Yaskawa INFORM job: SKRZYNIA_5040_180_STOPNI_20BR.JBI

/JOB
//NAME SKRZYNIA_5040_180_STOPNI_20BR
///FOLDERNAME 02-SKRZYNIE_JOBS
//POS
///NPOS 317,317,0,20,0,0
///TOOL 0
///POSTYPE PULSE
///PULSE
C00000=2424,-36726,63513,-9090,2744,5131
C00001=17840,-61498,-6635,149088,-29435,16513
C00002=84284,-61498,-6635,149088,14842,16513
C00003=84426,-61498,-62039,149088,14842,16513
C00004=84426,-61498,-83719,149088,14842,16513
C00005=79414,-27317,-83719,149088,18958,2543
C00006=73372,-22345,-79926,156833,908,-5737
C00007=69654,-19285,-77591,161600,-10201,-10832
C00008=80044,-19258,-92768,151274,-43492,-95
C00009=80167,-17748,-91560,151286,-43793,-146
C00010=77855,-16084,-90189,153542,-43693,-832
C00011=79745,-14573,-88908,151903,-44240,-404
C00012=80167,-17748,-91560,151286,-43793,-146
C00013=69654,-19285,-77591,161600,-10201,-10832
C00014=57344,-27370,-54568,135214,21884,-6631
C00015=40625,-29987,-49847,90639,36967,7668
C00016=40625,-29987,-49847,90639,36967,7668
C00017=38826,-24689,-45962,89185,38103,8693
C00018=37513,-22163,-43982,88710,38957,9107
C00019=39668,-21791,-43686,88310,37528,9139
C00020=38826,-24689,-45962,89185,38103,8693
C00021=38826,-24689,-45962,89185,38103,8693
C00022=42409,-29700,-46133,101604,34212,3947
C00023=39533,-32421,-42056,71487,38902,9246
C00024=48036,-29192,-45512,38244,44119,19118
C00025=48294,-22040,-40120,37064,45319,19886
C00026=46721,-19694,-38209,37780,46327,19540
C00027=48498,-19279,-37864,36630,45652,20159
C00028=48294,-22040,-40120,37064,45319,19886
C00029=39533,-32421,-42056,71487,38902,9246
C00030=80982,-65498,-53595,111483,16829,-11863
C00031=83918,-61953,-48743,149551,29621,-25735
C00032=40577,-31455,-39147,101508,36831,1521
C00033=62120,-15586,-68046,125419,11390,483
C00034=60388,-9931,-64401,116490,11174,5090
C00035=60671,-7045,-63303,110274,10395,8002
C00036=59274,-5305,-61557,108886,11033,8950
C00037=60834,-4584,-60819,109690,10258,8249
C00038=60671,-7045,-63303,110274,10395,8002
C00039=63645,-11488,-68603,127053,9270,213
C00040=46424,-32589,-51504,107545,30005,2440
C00041=40681,-36168,-63553,67140,38442,15724
C00042=40938,-28250,-58216,64472,39150,17313
C00043=40029,-26609,-57013,64509,39850,17414
C00044=42034,-26290,-56776,63350,38705,17844
C00045=40938,-28250,-58216,64472,39150,17313
C00046=45508,-32760,-62864,41083,46895,21518
C00047=52894,-26615,-39300,28664,42870,21364
C00048=47235,-10440,-23632,29897,60724,24736
C00049=57477,-15037,-17222,22818,38920,22189
C00050=55882,-13164,-15543,23879,39595,21547
C00051=57525,-12586,-15014,22628,39205,22306
C00052=57477,-15037,-17222,22818,38920,22189
C00053=51366,-27458,-41337,29323,44055,21022
C00054=95860,-54197,-56233,-11506,28414,43359
C00055=86028,-64310,-60026,34123,6588,25352
C00056=86028,-64310,-60026,34123,6588,25352
C00057=40577,-31455,-39147,101508,36831,1521
C00058=51132,-28512,-40196,130224,31508,-6645
C00059=50713,-22313,-35527,128251,30719,-5539
C00060=49231,-20302,-33901,126844,31206,-4688
C00061=50925,-19906,-33576,127815,30296,-5311
C00062=50713,-22313,-35527,128251,30719,-5539
C00063=49451,-30533,-41612,129729,32711,-6303
C00064=40577,-31455,-39147,101508,36831,1521
C00065=40577,-27956,-24714,110033,39226,-3600
C00066=40286,-31815,-40383,67790,38842,9831
C00067=40401,-25839,-36160,65987,39341,10928
C00068=39238,-23870,-34666,65921,40243,11019
C00069=41502,-23454,-34345,64975,38856,11500
C00070=40401,-25839,-36160,65987,39341,10928
C00071=40577,-31455,-39147,101508,36831,1521
C00072=86028,-64310,-60026,34123,6588,25352
C00073=86028,-64310,-60026,57978,24772,25352
C00074=86028,-64309,-60028,57978,24769,25352
C00075=40577,-31455,-39147,101508,36831,1521
C00076=38903,-31338,-35872,81629,38108,5349
C00077=39925,-26217,-33347,78892,37684,6977
C00078=38254,-23236,-30426,78887,38846,7020
C00079=40125,-23024,-30182,78580,37583,7157
C00080=39925,-26217,-33347,78892,37684,6977
C00081=73009,-49204,-27678,59140,12738,9351
C00082=45844,-59376,-6382,28358,16063,-8083
C00083=0,-52280,40443,0,6876,0
C00084=0,-39497,64868,0,-320,0
C00085=-26447,-43949,27117,-136096,-23097,-25575
C00086=-84284,-61498,-6635,-149088,14842,-16513
C00087=-84426,-61498,-62039,-149088,14842,-16513
C00088=-84426,-61498,-83719,-149088,14842,-16513
C00089=-80044,-19258,-92768,-151274,-43492,95
C00090=-80749,-16896,-90804,-150801,-44007,28
C00091=-79084,-15727,-89832,-152410,-43912,514
C00092=-80653,-14642,-88911,-151047,-44347,160
C00093=-80749,-16896,-90804,-150801,-44007,28
C00094=-75682,-33870,-78741,-101873,-8535,-10935
C00095=-48995,-37760,-57128,-94978,29787,-5634
C00096=-40649,-29976,-49851,-90623,36950,-7675
C00097=-40649,-29976,-49851,-90623,36950,-7675
C00098=-40401,-23900,-45312,-88796,37053,-8777
C00099=-39435,-22127,-43911,-88459,37683,-9068
C00100=-40828,-22111,-43897,-88252,36759,-9057
C00101=-40401,-23900,-45312,-88796,37053,-8777
C00102=-38849,-24678,-45965,-89170,38087,-8700
C00103=-42432,-29691,-46140,-101591,34194,-3953
C00104=-39561,-32409,-42051,-71473,38885,-9254
C00105=-48061,-29176,-45495,-38229,44108,-19126
C00106=-49260,-20540,-32676,-39004,41808,-18545
C00107=-48004,-18750,-31193,-39572,42610,-18251
C00108=-49371,-18582,-31053,-38688,42033,-18742
C00109=-49260,-20540,-32676,-39004,41808,-18545
C00110=-39561,-30849,-34727,-76036,37950,-6495
C00111=-96080,-64740,-46265,-152525,12897,30451
C00112=-81019,-62154,-45781,-119230,18197,15675
C00113=-39561,-30849,-34727,-76036,37950,-6495
C00114=-48406,-29556,-69320,-92179,25398,-12686
C00115=-47328,-23620,-66389,-87519,25941,-15295
C00116=-49848,-19619,-64817,-82594,24521,-17422
C00117=-48924,-18187,-63619,-82477,25084,-17649
C00118=-50351,-17944,-63415,-81734,24256,-17779
C00119=-49848,-19619,-64817,-82594,24521,-17422
C00120=-49519,-27286,-70984,-91916,23952,-13794
C00121=-40751,-34689,-48106,-81426,35657,-8146
C00122=-40681,-36168,-63553,-67140,38442,-15724
C00123=-43821,-29034,-57028,-64528,36876,-16908
C00124=-42088,-26142,-54916,-64622,38193,-17071
C00125=-43742,-25965,-54783,-63683,37230,-17421
C00126=-43821,-29034,-57028,-64528,36876,-16908
C00127=-45534,-32689,-56736,-43795,43869,-19675
C00128=-52916,-25303,-32096,-30881,39442,-19966
C00129=-58280,-19120,-27405,-20546,42356,-23593
C00130=-59518,-12125,-8161,-23315,34652,-21915
C00131=-57886,-10293,-6452,-24525,35301,-21178
C00132=-59048,-10070,-6241,-23572,34987,-21754
C00133=-59518,-12125,-8161,-23315,34652,-21915
C00134=-51388,-26224,-34221,-31487,40653,-19631
C00135=-51388,-26224,-34221,-31487,40653,-19631
C00136=-88798,-58761,-51280,2265,16070,-39336
C00137=-86028,-64310,-60026,-34123,6588,-25352
C00138=-40577,-31455,-39147,-101508,36831,-1521
C00139=-51132,-28512,-40196,-130224,31508,6645
C00140=-53828,-21538,-34856,-130236,29103,6776
C00141=-52017,-19235,-32968,-128427,29694,5703
C00142=-53263,-19086,-32845,-129254,29059,6216
C00143=-53828,-21538,-34856,-130236,29103,6776
C00144=-49451,-30533,-41612,-129729,32711,6303
C00145=-40577,-31455,-39147,-101508,36831,-1521
C00146=-40577,-27956,-24714,-110033,39226,3600
C00147=-40286,-31815,-40383,-67790,38842,-9831
C00148=-43936,-25540,-35936,-64541,37153,-11660
C00149=-42305,-23005,-33995,-64547,38400,-11722
C00150=-43835,-22890,-33904,-63890,37459,-12051
C00151=-43936,-25540,-35936,-64541,37153,-11660
C00152=-40577,-31455,-39147,-101508,36831,-1521
C00153=-86028,-64310,-60026,-34123,6588,-25352
C00154=-86028,-64310,-60026,-57978,24772,-25352
C00155=-86028,-64309,-60028,-57978,24769,-25352
C00156=-38903,-32774,-42709,-77257,38620,-7991
C00157=-42184,-24671,-30182,-79828,36015,-6379
C00158=-40569,-22194,-28667,-79025,37222,-6883
C00159=-42422,-21657,-27035,-79658,35870,-6476
C00160=-42184,-24671,-30182,-79828,36015,-6379
C00161=-49485,-27068,-14424,-72878,29346,-3454
C00162=-73009,-40277,-6382,-95546,11240,8083
C00163=-45844,-59376,-6382,-28358,16063,8083
C00164=0,-52280,40443,0,6876,0
C00165=-328,-40297,61840,-3808,1166,2006
C00166=17840,-61498,-6635,149088,-29435,16513
C00167=84284,-61498,-6635,149088,14842,16513
C00168=84513,-69641,-44219,158038,21366,7151
C00169=47085,-54494,-58070,115522,48054,-5105
C00170=38967,-30574,-72694,69596,39131,19833
C00171=38967,-30574,-72694,69596,39131,19833
C00172=40878,-31428,-43525,94415,35447,4548
C00173=41854,-23003,-37366,91536,34575,6162
C00174=41898,-23706,-43940,85918,34440,9382
C00175=40878,-31428,-43525,94415,35447,4548
C00176=39533,-30860,-34732,76047,37967,6488
C00177=46634,-28948,-39362,44629,40673,16329
C00178=47197,-19209,-31862,42612,41940,17576
C00179=47198,-18019,-24610,45914,39068,15513
C00180=46634,-28948,-39362,44629,40673,16329
C00181=49331,-35046,-41363,50989,36464,13786
C00182=89354,-53419,-27647,126582,13574,2293
C00183=87455,-53096,-27566,122620,14401,3981
C00184=17840,-61498,-6635,149088,-29435,16513
C00185=0,-40660,62594,0,368,0
C00186=-17840,-45374,24451,-139252,-21484,-21626
C00187=-84284,-61498,-6635,-149088,14842,-16513
C00188=-72689,-59179,-38530,-131034,19974,-20147
C00189=-60772,-50498,-67929,-131953,39604,8737
C00190=-35436,-23032,-76859,-79659,38842,-23552
C00191=-45272,-23185,-79217,-69622,29986,-24621
C00192=-40692,-30585,-47134,-93878,35604,-6100
C00193=-40001,-32873,-51156,-81642,36602,-9590
C00194=-40001,-32873,-51156,-81642,36602,-9590
C00195=-40670,-20516,-31954,-95909,37519,2638
C00196=-40659,-21415,-38860,-90776,37084,-418
C00197=-40001,-32873,-51156,-81642,36602,-9590
C00198=-40870,-31947,-42232,-63836,39356,-11267
C00199=-49698,-28191,-44773,-34393,44991,-20180
C00200=-50470,-17992,-36746,-32748,46471,-21232
C00201=-50479,-17271,-29967,-35030,43083,-19704
C00202=-49698,-28191,-44773,-34393,44991,-20180
C00203=-49698,-28786,-61181,-29564,54118,-23727
C00204=-82387,-65169,-54524,-93566,14000,4306
C00205=-84284,-61498,-6635,-149088,14842,-16513
C00206=-17840,-55538,4678,-146289,-26509,-18006
C00207=0,-39879,64121,0,-95,0
C00208=0,-52280,40443,0,6876,0
C00209=0,-52279,40442,0,6873,-1
C00210=65212,-60046,-8049,104848,-4690,-17864
C00211=39533,-30860,-34732,76047,37967,6488
C00212=40614,-18402,-49700,108061,37841,3104
C00213=40614,-18402,-49700,108061,37841,3104
C00214=41485,-12828,-44769,107158,37037,3517
C00215=41606,-12003,-50092,101801,35658,6646
C00216=40614,-18402,-49700,108061,37841,3104
C00217=40614,-18402,-49700,108061,37841,3104
C00218=49502,-29076,-56400,114238,27233,2182
C00219=40723,-34700,-48106,81442,35674,8138
C00220=40409,-20441,-6217,113220,40048,-7375
C00221=42493,-16023,-2566,113375,38437,-7307
C00222=42407,-18778,-11657,108563,36754,-4436
C00223=40409,-20441,-6217,113220,40048,-7375
C00224=39142,-35162,-55050,69516,38837,12809
C00225=56371,-25167,-46588,19640,50472,24717
C00226=56370,-24708,-41585,20550,47569,24051
C00227=56918,-11874,-10453,25192,36609,21079
C00228=55886,-6496,-6457,23354,43942,22802
C00229=56370,-20008,-17514,26362,35642,20382
C00230=64715,-29320,-15625,38703,25818,15298
C00231=92185,-54275,-12566,86648,-10406,-3964
C00232=0,-52279,40442,0,6873,-1
C00233=0,-52279,40442,0,6873,1
C00234=-37964,-53933,3758,-67381,6079,8710
C00235=-49904,-54659,-13207,-92831,9076,10998
C00236=-40577,-31455,-39147,-101508,36831,-1521
C00237=-37616,-19376,-56763,-96336,39614,-8284
C00238=-37616,-19376,-56763,-96336,39614,-8284
C00239=-40511,-13581,-51709,-94759,37718,-8730
C00240=-40499,-12353,-56710,-89299,37353,-11996
C00241=-37616,-19376,-56763,-96336,39614,-8284
C00242=-29868,-22288,-62791,-69139,55102,-14753
C00243=-38799,-34785,-68031,-65062,42004,-17700
C00244=-40843,-35617,-55345,-69003,37714,-12979
C00245=-40440,-20436,-6228,-113223,40025,7374
C00246=-44187,-15892,-2555,-114126,37382,7633
C00247=-44098,-18576,-11485,-109220,35681,4746
C00248=-40440,-20436,-6228,-113223,40025,7374
C00249=-39177,-35147,-55048,-69491,38818,-12821
C00250=-56396,-25146,-46559,-19625,50462,-24726
C00251=-56395,-19986,-17482,-26346,35629,-20392
C00252=-58275,-11034,-9655,-24079,36290,-21752
C00253=-53190,-4481,-3595,-29275,45221,-22163
C00254=-57665,-14024,-8618,-26361,33798,-20418
C00255=-54116,-36015,-20945,-72642,23963,-3174
C00256=-66633,-56546,-10672,-107930,-1326,17731
C00257=0,-52279,40442,0,6873,1
C00258=1,-52278,40440,0,6869,2
C00259=71244,-62242,-42760,28259,6636,20995
C00260=86028,-64310,-60026,34123,6588,25352
C00261=40577,-31455,-39147,101508,36831,1521
C00262=59968,-20268,-35682,154489,33643,-14406
C00263=49575,-29432,-40732,125662,31704,-5163
C00264=49462,-20616,-33510,124217,30834,-4171
C00265=49522,-21549,-40421,118611,28458,-1132
C00266=49575,-29432,-40732,125662,31704,-5163
C00267=40577,-31455,-39147,101508,36831,1521
C00268=40577,-27956,-24714,110033,39226,-3600
C00269=40745,-32658,-46054,62068,40241,12517
C00270=41807,-24195,-39992,59384,40616,14125
C00271=41807,-23141,-33009,63548,38813,11557
C00272=40745,-32658,-46054,62068,40241,12517
C00273=40577,-31455,-39147,101508,36831,1521
C00274=86028,-64310,-60026,34123,6588,25352
C00275=71244,-62242,-42760,28259,6636,20995
C00276=1,-52278,40440,0,6869,2
C00277=-71244,-62242,-42760,-28259,6636,-20995
C00278=-86028,-64310,-60026,-34123,6588,-25352
C00279=-40577,-31455,-39147,-101508,36831,-1521
C00280=-59968,-20268,-35682,-154489,33643,14406
C00281=-49575,-29432,-40732,-125662,31704,5163
C00282=-51745,-20083,-33073,-125482,29566,4973
C00283=-51720,-20470,-39541,-119439,27111,1736
C00284=-49575,-29432,-40732,-125662,31704,5163
C00285=-40577,-31455,-39147,-101508,36831,-1521
C00286=-40577,-27956,-24714,-110033,39226,3600
C00287=-40745,-32658,-46054,-62068,40241,-12517
C00288=-43918,-23250,-39259,-58141,39481,-14752
C00289=-43886,-22328,-32371,-62491,37605,-12114
C00290=-40745,-32658,-46054,-62068,40241,-12517
C00291=-40577,-31455,-39147,-101508,36831,-1521
C00292=-86028,-64310,-60026,-34123,6588,-25352
C00293=-71244,-62242,-42760,-28259,6636,-20995
C00294=-1,-52278,40440,0,6869,-2
C00295=2,-52272,40438,1,6859,6
C00296=86028,-64309,-60028,57978,24769,25352
C00297=40577,-29271,-29688,107326,38311,-1954
C00298=39686,-18672,-6528,106229,39889,-5106
C00299=40115,-16641,-6285,104879,39175,-4249
C00300=40039,-18622,-13956,100467,38186,-1572
C00301=40578,-24372,-18301,102198,38163,-2598
C00302=51067,-26075,-7125,86189,26964,-2285
C00303=73009,-40277,-6382,95546,11240,-8083
C00304=45844,-59376,-6382,28358,16063,-8083
C00305=0,-52280,40443,0,6876,0
C00306=-49336,-60774,-21138,-33872,18352,-14728
C00307=-86028,-64309,-60028,-57978,24769,-25352
C00308=-40577,-31455,-39147,-101508,36831,-1521
C00309=-39686,-19839,-10359,-104288,39330,3911
C00310=-42399,-15880,-6496,-104843,37485,4096
C00311=-42423,-18479,-15943,-99204,36274,759
C00312=-40581,-27576,-30519,-94819,36955,-1807
C00313=-56174,-25706,-11107,-56673,25485,-9093
C00314=-73009,-40277,-6382,-95546,11240,8083
C00315=-45844,-59376,-6382,-28358,16063,8083
C00316=0,-52280,40443,0,6876,0
BC00000=467540
BC00001=467540
BC00002=467540
BC00003=467540
BC00004=467540
BC00005=467540
BC00006=467540
BC00007=467540
BC00008=467540
BC00009=467540
BC00010=467540
BC00011=467540
BC00012=467540
BC00013=467540
BC00014=507878
BC00015=487125
BC00016=487125
BC00017=487125
BC00018=487125
BC00019=487125
BC00020=487125
BC00021=487125
BC00022=485653
BC00023=485653
BC00024=485653
BC00025=485653
BC00026=485653
BC00027=485653
BC00028=485653
BC00029=485653
BC00030=485653
BC00031=675626
BC00032=675626
BC00033=714617
BC00034=714617
BC00035=714617
BC00036=714617
BC00037=714617
BC00038=714617
BC00039=717870
BC00040=686402
BC00041=686402
BC00042=686402
BC00043=686402
BC00044=686402
BC00045=686402
BC00046=655680
BC00047=655680
BC00048=655680
BC00049=655680
BC00050=655680
BC00051=655680
BC00052=655680
BC00053=612974
BC00054=633023
BC00055=817027
BC00056=849627
BC00057=849627
BC00058=849627
BC00059=849627
BC00060=849627
BC00061=849627
BC00062=849627
BC00063=849627
BC00064=849627
BC00065=849627
BC00066=849627
BC00067=849627
BC00068=849627
BC00069=849627
BC00070=849627
BC00071=849627
BC00072=849627
BC00073=849627
BC00074=994223
BC00075=997528
BC00076=995174
BC00077=996484
BC00078=995671
BC00079=995573
BC00080=996484
BC00081=965704
BC00082=879640
BC00083=828403
BC00084=484492
BC00085=467540
BC00086=467540
BC00087=467540
BC00088=467540
BC00089=467540
BC00090=467542
BC00091=467542
BC00092=467542
BC00093=467542
BC00094=476933
BC00095=486269
BC00096=487125
BC00097=487125
BC00098=487125
BC00099=487125
BC00100=487125
BC00101=487125
BC00102=487125
BC00103=485653
BC00104=485653
BC00105=485653
BC00106=477973
BC00107=477973
BC00108=477973
BC00109=477973
BC00110=477973
BC00111=477973
BC00112=637224
BC00113=637224
BC00114=676215
BC00115=676215
BC00116=676215
BC00117=676215
BC00118=676215
BC00119=676215
BC00120=679468
BC00121=648000
BC00122=686402
BC00123=686402
BC00124=686402
BC00125=686402
BC00126=686402
BC00127=648000
BC00128=648000
BC00129=648000
BC00130=648000
BC00131=648000
BC00132=648000
BC00133=648000
BC00134=648000
BC00135=624365
BC00136=626985
BC00137=849627
BC00138=849627
BC00139=849627
BC00140=849627
BC00141=849627
BC00142=849627
BC00143=849627
BC00144=849627
BC00145=849627
BC00146=849627
BC00147=849627
BC00148=849627
BC00149=849627
BC00150=849627
BC00151=849627
BC00152=849627
BC00153=849627
BC00154=849627
BC00155=994094
BC00156=1002378
BC00157=995010
BC00158=995501
BC00159=994027
BC00160=995010
BC00161=965704
BC00162=944514
BC00163=879640
BC00164=828403
BC00165=489545
BC00166=498510
BC00167=467540
BC00168=484470
BC00169=489677
BC00170=489675
BC00171=489675
BC00172=477973
BC00173=477973
BC00174=477973
BC00175=477973
BC00176=477973
BC00177=477973
BC00178=477973
BC00179=477973
BC00180=477973
BC00181=458600
BC00182=448949
BC00183=525722
BC00184=487426
BC00185=486611
BC00186=479113
BC00187=467540
BC00188=470459
BC00189=528079
BC00190=528079
BC00191=528077
BC00192=477973
BC00193=477973
BC00194=477973
BC00195=477973
BC00196=477973
BC00197=477973
BC00198=477973
BC00199=477973
BC00200=477973
BC00201=477973
BC00202=477973
BC00203=477973
BC00204=477973
BC00205=467540
BC00206=467540
BC00207=482699
BC00208=527850
BC00209=541981
BC00210=560285
BC00211=642547
BC00212=672480
BC00213=672480
BC00214=672480
BC00215=672480
BC00216=672480
BC00217=672480
BC00218=679468
BC00219=648000
BC00220=648000
BC00221=648000
BC00222=648000
BC00223=648000
BC00224=648000
BC00225=648000
BC00226=648000
BC00227=648000
BC00228=648000
BC00229=607087
BC00230=565122
BC00231=563264
BC00232=528036
BC00233=500175
BC00234=526377
BC00235=553881
BC00236=649161
BC00237=672480
BC00238=672480
BC00239=672480
BC00240=672480
BC00241=672480
BC00242=634078
BC00243=641066
BC00244=648000
BC00245=648000
BC00246=648000
BC00247=648000
BC00248=648000
BC00249=648000
BC00250=648000
BC00251=608255
BC00252=648000
BC00253=648000
BC00254=613281
BC00255=601855
BC00256=554421
BC00257=532052
BC00258=574254
BC00259=802302
BC00260=849627
BC00261=849627
BC00262=849627
BC00263=849627
BC00264=849627
BC00265=849627
BC00266=849627
BC00267=849627
BC00268=849627
BC00269=849627
BC00270=849627
BC00271=849627
BC00272=849627
BC00273=849627
BC00274=849627
BC00275=802302
BC00276=652677
BC00277=802302
BC00278=849627
BC00279=849627
BC00280=849627
BC00281=849627
BC00282=849627
BC00283=849627
BC00284=849627
BC00285=849627
BC00286=849627
BC00287=849627
BC00288=849627
BC00289=849627
BC00290=849627
BC00291=849627
BC00292=849627
BC00293=802302
BC00294=652677
BC00295=780547
BC00296=1007134
BC00297=993409
BC00298=989933
BC00299=991571
BC00300=991571
BC00301=990663
BC00302=974575
BC00303=965704
BC00304=879640
BC00305=828403
BC00306=894245
BC00307=994909
BC00308=994105
BC00309=993208
BC00310=992554
BC00311=992554
BC00312=984659
BC00313=957065
BC00314=965704
BC00315=879640
BC00316=828403
///POSTYPE BASE
///RECTAN
///RCONF 1,0,0,0,0,0,0,0,0,0,0,0,0,0,0,0,0,0,0,0,0,0,0,0
P00006=0.000,0.000,0.000,0.0000,0.0000,0.0000
///RCONF 0,0,0,0,0,0,0,0,0,0,0,0,0,0,0,0,0,0,0,0,0,0,0,0
P00056=0.000,0.000,5.000,0.0000,0.0000,0.0000
///RCONF 1,0,0,0,0,0,0,0,0,0,0,0,0,0,0,0,0,0,0,0,0,0,0,0
P00300=-0.036,-1.505,2.318,0.0000,0.0000,0.0000
P00301=0.028,-0.041,7.752,0.0000,0.0000,0.0000
///RCONF 0,0,0,0,0,0,0,0,0,0,0,0,0,0,0,0,0,0,0,0,0,0,0,0
P00302=0.052,-2.937,-4.426,0.0000,0.0000,0.0000
P00303=-0.004,-1.437,-4.584,0.0000,0.0000,0.0000
P00304=0.028,-1.666,-4.234,0.0000,0.0000,0.0000
P00305=-0.003,-1.920,-3.501,0.0000,0.0000,0.0000
P00306=0.015,-2.252,-3.054,0.0000,0.0000,0.0000
P00307=0.019,-2.151,-5.077,0.0000,0.0000,0.0000
P00308=-0.003,-2.092,-4.888,0.0000,0.0000,0.0000
P00350=11.519,-0.008,1.149,0.0000,0.0000,0.0000
P00351=13.563,-0.027,-0.653,0.0000,0.0000,0.0000
P00352=13.252,-0.027,-0.827,0.0000,0.0000,0.0000
P00353=10.971,-0.082,0.776,0.0000,0.0000,0.0000
P00354=-0.024,2.508,-1.824,0.0000,0.0000,0.0000
P00355=-0.001,2.528,-1.131,0.0000,0.0000,0.0000
P00356=-0.034,2.921,-0.262,0.0000,0.0000,0.0000
P00357=0.003,3.386,-0.091,0.0000,0.0000,0.0000
P00358=0.014,3.037,-0.020,0.0000,0.0000,0.0000
//INST
///DATE 2024/05/16 17:47
///ATTR SC,RW
///GROUP1 RB1,BS1
NOP
CALL JOB:MOVE_INTO_TUNNEL
MOVJ C00000 BC00000 VJ=10.00
MOVJ C00001 BC00001 VJ=10.00
MOVJ C00002 BC00002 VJ=10.00
MOVJ C00003 BC00003 VJ=10.00
MOVJ C00004 BC00004 VJ=10.00
MOVJ C00005 BC00005 VJ=10.00
MOVJ C00006 BC00006 VJ=10.00
MOVL C00007 BC00007 V=150.0
MOVL C00008 BC00008 V=150.0
'------------------------
'W63.3
'------------------------
MOVL C00009 BC00009 V=66.7 PL=0
REFP 3 C00010 BC00010
CALL JOB:SEARCH-R1
IMOV P0056 V=23.0
SET P0300 P0006
SFTON P0300
REFP 3 C00011 BC00011
CALL JOB:SEARCH-R1
SET P0300 P0006
SFTON P0300
MOVL C00012 BC00012 V=66.7 PL=0
SFTOF
'PRZEJAZD
MOVL C00013 BC00013 V=150.0
MOVL C00014 BC00014 V=666.7
MOVJ C00015 BC00015 VJ=10.00
MOVL C00016 BC00016 V=150.0
'------------------------
'W29.6
'------------------------
MOVL C00017 BC00017 V=66.7 PL=0
REFP 3 C00018 BC00018
CALL JOB:SEARCH-R1
IMOV P0056 V=23.0 PL=0
SET P0301 P0006
SFTON P0301
REFP 3 C00019 BC00019
CALL JOB:SEARCH-R1
SET P0301 P0006
SFTON P0301
MOVL C00020 BC00020 V=66.7 PL=0
SFTOF
'PRZEJAZD
MOVL C00021 BC00021 V=500.0
MOVL C00022 BC00022 V=500.0
MOVL C00023 BC00023 V=500.0
MOVL C00024 BC00024 V=500.0
'------------------------
'W29.9
'------------------------
MOVL C00025 BC00025 V=66.7 PL=0
REFP 3 C00026 BC00026
CALL JOB:SEARCH-R1
IMOV P0056 V=23.0 PL=0
SET P0302 P0006
SFTON P0302
REFP 3 C00027 BC00027
CALL JOB:SEARCH-R1
SET P0302 P0006
SFTON P0302
MOVL C00028 BC00028 V=66.7 PL=0
SFTOF
MOVL C00029 BC00029 V=500.0
'PRZEJAZD
MOVL C00030 BC00030 V=500.0
MOVJ C00031 BC00031 VJ=10.00
MOVL C00032 BC00032 V=500.0
MOVL C00033 BC00033 V=500.0
MOVL C00034 BC00034 V=500.0
'------------------------
'W63.12
'------------------------
MOVL C00035 BC00035 V=66.7 PL=0
REFP 3 C00036 BC00036
CALL JOB:SEARCH-R1
IMOV P0056 V=23.0 PL=0
SET P0303 P0006
SFTON P0303
REFP 3 C00037 BC00037
CALL JOB:SEARCH-R1
SET P0303 P0006
SFTON P0303
MOVL C00038 BC00038 V=66.7 PL=0
SFTOF
'PRZEJAZD
MOVL C00039 BC00039 V=500.0
MOVL C00040 BC00040 V=500.0
MOVL C00041 BC00041 V=500.0
'------------------------
'W63.15
'------------------------
MOVL C00042 BC00042 V=66.7 PL=0
REFP 3 C00043 BC00043
CALL JOB:SEARCH-R1
IMOV P0056 V=23.0 PL=0
SET P0304 P0006
SFTON P0304
REFP 3 C00044 BC00044
CALL JOB:SEARCH-R1
SET P0304 P0006
SFTON P0304
MOVL C00045 BC00045 V=66.7 PL=0
SFTOF
'PRZEJAZD
MOVL C00046 BC00046 V=500.0
MOVL C00047 BC00047 V=500.0
MOVL C00048 BC00048 V=500.0
'------------------------
'W29.18
'------------------------
MOVL C00049 BC00049 V=66.7 PL=0
REFP 3 C00050 BC00050
CALL JOB:SEARCH-R1
IMOV P0056 V=23.0 PL=0
SET P0305 P0006
SFTON P0305
REFP 3 C00051 BC00051
CALL JOB:SEARCH-R1
SET P0305 P0006
SFTON P0305
MOVL C00052 BC00052 V=66.7 PL=0
SFTOF
'PRZEJAZD
MOVL C00053 BC00053 V=500.0
MOVJ C00054 BC00054 VJ=10.00
MOVJ C00055 BC00055 VJ=10.00
MOVJ C00056 BC00056 VJ=10.00
MOVL C00057 BC00057 V=500.0
MOVL C00058 BC00058 V=500.0
'------------------------
'W29.21
'------------------------
MOVL C00059 BC00059 V=66.7 PL=0
REFP 3 C00060 BC00060
CALL JOB:SEARCH-R1
IMOV P0056 V=23.0 PL=0
SET P0306 P0006
SFTON P0306
REFP 3 C00061 BC00061
CALL JOB:SEARCH-R1
SET P0306 P0006
SFTON P0306
MOVL C00062 BC00062 V=66.7 PL=0
SFTOF
'PRZEJAZD
MOVL C00063 BC00063 V=500.0
MOVL C00064 BC00064 V=500.0
MOVL C00065 BC00065 V=500.0
MOVL C00066 BC00066 V=500.0
'------------------------
'W29.24
'------------------------
MOVL C00067 BC00067 V=66.7 PL=0
REFP 3 C00068 BC00068
CALL JOB:SEARCH-R1
IMOV P0056 V=23.0 PL=0
SET P0307 P0006
SFTON P0307
REFP 3 C00069 BC00069
CALL JOB:SEARCH-R1
SET P0307 P0006
SFTON P0307
MOVL C00070 BC00070 V=66.7 PL=0
SFTOF
'PRZEJAZD
MOVL C00071 BC00071 V=500.0
MOVL C00072 BC00072 V=500.0
MOVL C00073 BC00073 V=500.0
MOVL C00074 BC00074 V=500.0
MOVL C00075 BC00075 V=500.0
MOVL C00076 BC00076 V=500.0
'BRAK MOZLIWOSCI 29.27
'BRAK MOZLIWOSCI 29.27
'BRAK MOZLIWOSCI 29.27
'BRAK MOZLIWOSCI 29.27
'BRAK MOZLIWOSCI 29.27
'------------------------
'W63.30
'------------------------
MOVL C00077 BC00077 V=166.7 PL=0
REFP 3 C00078 BC00078
CALL JOB:SEARCH-R1
IMOV P0056 V=23.0 PL=0
SET P0308 P0006
SFTON P0308
REFP 3 C00079 BC00079
CALL JOB:SEARCH-R1
SET P0308 P0006
SFTON P0308
MOVL C00080 BC00080 V=250.0 PL=0
SFTOF
'PRZEJAZD
MOVJ C00081 BC00081 VJ=20.00
MOVJ C00082 BC00082 VJ=30.00
MOVJ C00083 BC00083 VJ=30.00
MOVJ C00084 BC00084 VJ=40.00
MOVJ C00085 BC00085 VJ=20.00
MOVJ C00086 BC00086 VJ=20.00
MOVJ C00087 BC00087 VJ=20.00
MOVJ C00088 BC00088 VJ=20.00
MOVL C00089 BC00089 V=500.0
'------------------------
'W63.3
'------------------------
MOVL C00090 BC00090 V=66.7 PL=0
REFP 3 C00091 BC00091
CALL JOB:SEARCH-R1
IMOV P0056 V=23.0
SET P0350 P0006
SFTON P0350
REFP 3 C00092 BC00092
CALL JOB:SEARCH-R1
SET P0350 P0006
SFTON P0350
MOVL C00093 BC00093 V=66.7 PL=0
SFTOF
'PRZEJAZD
MOVL C00094 BC00094 V=150.0 PL=0
MOVJ C00095 BC00095 VJ=10.00
MOVJ C00096 BC00096 VJ=10.00
MOVL C00097 BC00097 V=150.0
'------------------------
'W29.6
'------------------------
MOVL C00098 BC00098 V=66.7 PL=0
REFP 3 C00099 BC00099
CALL JOB:SEARCH-R1
IMOV P0056 V=23.0 PL=0
SET P0351 P0006
SFTON P0351
REFP 3 C00100 BC00100
CALL JOB:SEARCH-R1
SET P0351 P0006
SFTON P0351
MOVL C00101 BC00101 V=66.7 PL=0
SFTOF
'PRZEJAZD
MOVL C00102 BC00102 V=500.0
MOVL C00103 BC00103 V=500.0
MOVL C00104 BC00104 V=500.0
MOVL C00105 BC00105 V=500.0
'------------------------
'W29.9
'------------------------
MOVL C00106 BC00106 V=66.7 PL=0
REFP 3 C00107 BC00107
CALL JOB:SEARCH-R1
IMOV P0056 V=23.0 PL=0
SET P0352 P0006
SFTON P0352
REFP 3 C00108 BC00108
CALL JOB:SEARCH-R1
SET P0352 P0006
SFTON P0352
MOVL C00109 BC00109 V=66.7 PL=0
SFTOF
MOVL C00110 BC00110 V=500.0
'PRZEJAZD
MOVL C00111 BC00111 V=500.0
MOVJ C00112 BC00112 VJ=30.00
MOVL C00113 BC00113 V=500.0
MOVL C00114 BC00114 V=500.0
MOVL C00115 BC00115 V=500.0
'------------------------
'W63.12
'------------------------
MOVL C00116 BC00116 V=66.7 PL=0
REFP 3 C00117 BC00117
CALL JOB:SEARCH-R1
IMOV P0056 V=23.0 PL=0
SET P0353 P0006
SFTON P0353
REFP 3 C00118 BC00118
CALL JOB:SEARCH-R1
SET P0353 P0006
SFTON P0353
MOVL C00119 BC00119 V=66.7 PL=0
SFTOF
'PRZEJAZD
MOVL C00120 BC00120 V=500.0
MOVL C00121 BC00121 V=500.0
MOVL C00122 BC00122 V=500.0
'------------------------
'W63.15
'------------------------
MOVL C00123 BC00123 V=66.7 PL=0
REFP 3 C00124 BC00124
CALL JOB:SEARCH-R1
IMOV P0056 V=23.0 PL=0
SET P0354 P0006
SFTON P0354
REFP 3 C00125 BC00125
CALL JOB:SEARCH-R1
SET P0354 P0006
SFTON P0354
MOVL C00126 BC00126 V=66.7 PL=0
SFTOF
'PRZEJAZD
MOVL C00127 BC00127 V=500.0
MOVL C00128 BC00128 V=500.0
MOVL C00129 BC00129 V=500.0
'------------------------
'W29.18
'------------------------
MOVL C00130 BC00130 V=66.7 PL=0
REFP 3 C00131 BC00131
CALL JOB:SEARCH-R1
IMOV P0056 V=23.0 PL=0
SET P0355 P0006
SFTON P0355
REFP 3 C00132 BC00132
CALL JOB:SEARCH-R1
SET P0355 P0006
SFTON P0355
MOVL C00133 BC00133 V=66.7 PL=0
SFTOF
'PRZEJAZD
MOVL C00134 BC00134 V=500.0
MOVJ C00135 BC00135 VJ=10.00
MOVJ C00136 BC00136 VJ=10.00
MOVJ C00137 BC00137 VJ=30.00
MOVL C00138 BC00138 V=500.0
MOVL C00139 BC00139 V=500.0
'------------------------
'W29.21
'------------------------
MOVL C00140 BC00140 V=66.7 PL=0
REFP 3 C00141 BC00141
CALL JOB:SEARCH-R1
IMOV P0056 V=23.0 PL=0
SET P0356 P0006
SFTON P0356
REFP 3 C00142 BC00142
CALL JOB:SEARCH-R1
SET P0356 P0006
SFTON P0356
MOVL C00143 BC00143 V=66.7 PL=0
SFTOF
'PRZEJAZD
MOVL C00144 BC00144 V=500.0
MOVL C00145 BC00145 V=500.0
MOVL C00146 BC00146 V=500.0
MOVL C00147 BC00147 V=500.0
'------------------------
'W29.24
'------------------------
MOVL C00148 BC00148 V=66.7 PL=0
REFP 3 C00149 BC00149
CALL JOB:SEARCH-R1
IMOV P0056 V=23.0 PL=0
SET P0357 P0006
SFTON P0357
REFP 3 C00150 BC00150
CALL JOB:SEARCH-R1
SET P0357 P0006
SFTON P0357
MOVL C00151 BC00151 V=66.7 PL=0
SFTOF
'PRZEJAZD
MOVL C00152 BC00152 V=500.0
MOVL C00153 BC00153 V=500.0
MOVL C00154 BC00154 V=500.0
MOVL C00155 BC00155 V=500.0
MOVL C00156 BC00156 V=500.0
'BRAK MOZLIWOSCI 29.27
'BRAK MOZLIWOSCI 29.27
'BRAK MOZLIWOSCI 29.27
'BRAK MOZLIWOSCI 29.27
'BRAK MOZLIWOSCI 29.27
'------------------------
'W63.30
'------------------------
MOVL C00157 BC00157 V=66.7 PL=0
REFP 3 C00158 BC00158
CALL JOB:SEARCH-R1
IMOV P0056 V=23.0 PL=0
SET P0358 P0006
SFTON P0358
REFP 3 C00159 BC00159
CALL JOB:SEARCH-R1
SET P0358 P0006
SFTON P0358
MOVL C00160 BC00160 V=66.7 PL=0
SFTOF
'PRZEJAZD
MOVL C00161 BC00161 V=500.0
MOVJ C00162 BC00162 VJ=30.00
MOVJ C00163 BC00163 VJ=30.00
MOVJ C00164 BC00164 VJ=30.00
MOVJ C00165 BC00165 VJ=30.00
MOVJ C00166 BC00166 VJ=20.00
MOVJ C00167 BC00167 VJ=20.00
MOVJ C00168 BC00168 VJ=20.00
MOVJ C00169 BC00169 VJ=20.00
SFTOF
'------------------------
'W63.3
'------------------------
'PRZEJAZD
MOVL C00170 BC00170 V=500.0
MOVL C00171 BC00171 V=500.0
'------------------------
'W29.6
'------------------------
MOVL C00172 BC00172 V=500.0
SFTON P0301
MOVL C00173 BC00173 V=166.7 PL=0
MACRO1 MJ#(0) ARGF24
ARCON
MOVL C00174 BC00174 V=10.8
ARCOF
SFTOF
MOVL C00175 BC00175 V=500.0
SFTOF
MOVL C00176 BC00176 V=500.0
'------------------------
'W29.9
'------------------------
MOVL C00177 BC00177 V=500.0
SFTON P0302
MOVL C00178 BC00178 V=66.7 PL=0
MACRO1 MJ#(0) ARGF24
ARCON
MOVL C00179 BC00179 V=10.8
ARCOF
SFTOF
MOVL C00180 BC00180 V=500.0
SFTOF
'PRZEJAZD
MOVL C00181 BC00181 V=500.0
MOVJ C00182 BC00182 VJ=10.00
MOVJ C00183 BC00183 VJ=10.00
MOVJ C00184 BC00184 VJ=10.00
MOVJ C00185 BC00185 VJ=10.00
'TEST
'TEST
'TEST
MOVJ C00186 BC00186 VJ=30.00
MOVJ C00187 BC00187 VJ=10.00
MOVJ C00188 BC00188 VJ=10.00
MOVJ C00189 BC00189 VJ=20.00
MOVL C00190 BC00190 V=500.0
MOVL C00191 BC00191 V=500.0
MOVL C00192 BC00192 V=500.0
MOVL C00193 BC00193 V=500.0
'------------------------
'W28.6
'------------------------
MOVL C00194 BC00194 V=500.0
SFTON P0351
MOVL C00195 BC00195 V=166.7 PL=0
MACRO1 MJ#(0) ARGF24
ARCON
MOVL C00196 BC00196 V=10.8
ARCOF
SFTOF
MOVL C00197 BC00197 V=500.0
SFTOF
MOVL C00198 BC00198 V=500.0
'------------------------
'W28.9
'------------------------
MOVL C00199 BC00199 V=500.0
SFTON P0352
MOVL C00200 BC00200 V=66.7 PL=0
MACRO1 MJ#(0) ARGF24
ARCON
MOVL C00201 BC00201 V=10.0
ARCOF
SFTOF
MOVL C00202 BC00202 V=500.0
SFTOF
'PRZEJAZD
MOVL C00203 BC00203 V=666.7
MOVL C00204 BC00204 V=500.0
MOVJ C00205 BC00205 VJ=10.00
MOVJ C00206 BC00206 VJ=10.00
MOVJ C00207 BC00207 VJ=20.00
MOVJ C00208 BC00208 VJ=30.00
MOVJ C00209 BC00209 VJ=30.00
MOVJ C00210 BC00210 VJ=20.00
MOVJ C00211 BC00211 VJ=20.00
'------------------------
'W63.12
'------------------------
MOVL C00212 BC00212 V=500.0
MOVL C00213 BC00213 V=66.7
SFTON P0303
MOVL C00214 BC00214 V=166.7 PL=0
ARCON
MOVL C00215 BC00215 V=10.0
ARCOF
SFTOF
MOVL C00216 BC00216 V=250.0
'PRZEJAZD
MOVL C00217 BC00217 V=500.0
MOVL C00218 BC00218 V=500.0
MOVL C00219 BC00219 V=500.0
'------------------------
'W63.15
'------------------------
MOVL C00220 BC00220 V=166.7
SFTON P0304
MOVL C00221 BC00221 V=166.7 PL=0
MACRO1 MJ#(0) ARGF24
ARCON
MOVL C00222 BC00222 V=10.0
ARCOF
SFTOF
MOVL C00223 BC00223 V=250.0
SFTOF
'PRZEJAZD
MOVL C00224 BC00224 V=500.0
MOVL C00225 BC00225 V=500.0
'------------------------
'W29.18
'------------------------
MOVL C00226 BC00226 V=66.7
SFTON P0305
MOVL C00227 BC00227 V=166.7 PL=0
ARCON
MOVL C00228 BC00228 V=10.0
ARCOF
SFTOF
MOVL C00229 BC00229 V=666.7
SFTOF
'PRZEJAZD
MOVJ C00230 BC00230 VJ=30.00
MOVJ C00231 BC00231 VJ=30.00
MOVJ C00232 BC00232 VJ=30.00
'COMMENT
'COMMENT
'COMMENT
'COMMENT
'COMMENT
MOVJ C00233 BC00233 VJ=30.00
MOVJ C00234 BC00234 VJ=30.00
MOVJ C00235 BC00235 VJ=30.00
MOVJ C00236 BC00236 VJ=30.00
'------------------------
'W62.12
'------------------------
MOVL C00237 BC00237 V=500.0
MOVL C00238 BC00238 V=166.7
SFTON P0353
MOVL C00239 BC00239 V=166.7 PL=0
ARCON
MOVL C00240 BC00240 V=10.0
ARCOF
SFTOF
MOVL C00241 BC00241 V=166.7
'PRZEJAZD
MOVL C00242 BC00242 V=500.0
MOVL C00243 BC00243 V=500.0
MOVL C00244 BC00244 V=500.0
'------------------------
'W62.15
'------------------------
MOVL C00245 BC00245 V=250.0
SFTON P0354
MOVL C00246 BC00246 V=166.7 PL=0
ARCON
MOVL C00247 BC00247 V=10.0
ARCOF
SFTOF
MOVL C00248 BC00248 V=250.0
SFTOF
'PRZEJAZD
MOVL C00249 BC00249 V=500.0
MOVL C00250 BC00250 V=500.0
'------------------------
'W28.18
'------------------------
MOVL C00251 BC00251 V=166.7
SFTON P0355
MOVL C00252 BC00252 V=166.7 PL=0
ARCON
MOVL C00253 BC00253 V=10.0
ARCOF
SFTOF
MOVL C00254 BC00254 V=666.7
SFTOF
'PRZEJAZD
MOVJ C00255 BC00255 VJ=30.00
MOVJ C00256 BC00256 VJ=30.00
MOVJ C00257 BC00257 VJ=30.00
MOVJ C00258 BC00258 VJ=30.00
MOVJ C00259 BC00259 VJ=30.00
MOVJ C00260 BC00260 VJ=30.00
MOVL C00261 BC00261 V=500.0
MOVL C00262 BC00262 V=500.0
'------------------------
'W63.21
'------------------------
MOVL C00263 BC00263 V=500.0
SFTON P0306
MOVL C00264 BC00264 V=166.7 PL=0
MACRO1 MJ#(0) ARGF24
ARCON
MOVL C00265 BC00265 V=10.0
ARCOF
SFTOF
MOVL C00266 BC00266 V=500.0
'PRZEJAZD
MOVL C00267 BC00267 V=500.0
MOVL C00268 BC00268 V=500.0
'------------------------
'W29.24
'------------------------
MOVL C00269 BC00269 V=500.0
SFTON P0307
MOVL C00270 BC00270 V=166.7 PL=0
MACRO1 MJ#(0) ARGF24
ARCON
MOVL C00271 BC00271 V=10.0
ARCOF
SFTOF
MOVL C00272 BC00272 V=500.0
SFTOF
'PRZEJAZD
'BRAK 29.26
'BRAK 29.26
'BRAK 29.26
'BRAK 29.26
'BRAK 29.26
'BRAK 29.26
MOVL C00273 BC00273 V=500.0
MOVJ C00274 BC00274 VJ=30.00
MOVJ C00275 BC00275 VJ=30.00
MOVJ C00276 BC00276 VJ=20.00
'TEST
'TEST
'TEST
'TEST
MOVJ C00277 BC00277 VJ=20.00
MOVJ C00278 BC00278 VJ=20.00
MOVL C00279 BC00279 V=500.0
MOVL C00280 BC00280 V=500.0
'------------------------
'W63.21
'------------------------
MOVL C00281 BC00281 V=500.0
SFTON P0306
MOVL C00282 BC00282 V=66.7 PL=0
ARCON
MOVL C00283 BC00283 V=10.0
ARCOF
SFTOF
MOVL C00284 BC00284 V=500.0
'PRZEJAZD
MOVL C00285 BC00285 V=500.0
MOVL C00286 BC00286 V=500.0
'------------------------
'W29.24
'------------------------
MOVL C00287 BC00287 V=500.0
SFTON P0307
MOVL C00288 BC00288 V=166.7 PL=0
ARCON
MOVL C00289 BC00289 V=10.0
ARCOF
SFTOF
MOVL C00290 BC00290 V=500.0
SFTOF
'PRZEJAZD
'BRAK 29.26
'BRAK 29.26
'BRAK 29.26
'BRAK 29.26
'BRAK 29.26
'BRAK 29.26
MOVL C00291 BC00291 V=500.0
MOVJ C00292 BC00292 VJ=20.00
MOVJ C00293 BC00293 VJ=20.00
MOVJ C00294 BC00294 VJ=20.00
MOVJ C00295 BC00295 VJ=20.00
MOVJ C00296 BC00296 VJ=30.00
MOVJ C00297 BC00297 VJ=30.00
'W29.27
'W29.27
'W29.27
'W29.27
'DO DOPISANIA NA GOTOWO
'------------------------
'W63.30
'------------------------
MOVL C00298 BC00298 V=166.7
SFTON P0308
MOVL C00299 BC00299 V=166.7 PL=0
ARCON
MOVL C00300 BC00300 V=10.0
ARCOF
SFTOF
MOVL C00301 BC00301 V=250.0
SFTOF
MOVL C00302 BC00302 V=500.0
MOVJ C00303 BC00303 VJ=30.00
MOVJ C00304 BC00304 VJ=30.00
MOVJ C00305 BC00305 VJ=30.00
MOVJ C00306 BC00306 VJ=30.00
'TEST
MOVJ C00307 BC00307 VJ=20.00
MOVJ C00308 BC00308 VJ=20.00
'W29.27
'W29.27
'W29.27
'W29.27
'DO DOPISANIA NA GOTOWO
'------------------------
'W63.30
'------------------------
MOVL C00309 BC00309 V=66.7
SFTON P0358
MOVL C00310 BC00310 V=66.7 PL=0
ARCON
MOVL C00311 BC00311 V=10.0
ARCOF
SFTOF
MOVL C00312 BC00312 V=166.7
SFTOF
MOVL C00313 BC00313 V=500.0
MOVJ C00314 BC00314 VJ=20.00
MOVJ C00315 BC00315 VJ=20.00
MOVJ C00316 BC00316 VJ=30.00
CALL JOB:MOVE_OUT_OF_TUNNEL
END
